// TIA Portal V17 export
// export: Created 2023-06-23T18:33:40.54636Z, ExportSetting WithDefaults, DisplayName Totally Integrated Automation Portal, DisplayVersion V17, DisplayName TIA Portal Openness, DisplayVersion V17, DisplayName TIA Portal Version Control Interface, DisplayVersion V17, DisplayName STEP 7 Professional, DisplayVersion V17, DisplayName STEP 7 Safety, DisplayVersion V17, DisplayName WinCC Advanced / Unified PC, DisplayVersion V17
VAR_GLOBAL   // PLC tag table "23_ESP-EG1"
   "iESP-EG1" AT %I13.0 : Bool;
   "oESP-EG1" AT %Q12.3 : Bool;
END_VAR
